FUNCTION_BLOCK EM_Utilities EXTENDS EM_Base IMPLEMENTS I_EM_Utilities
VAR
	//Control modules
	s_diSafetyOk : FB_DigInput;
	s_diPowerOk : FB_DigInput;
	s_diAirPressureOk : FB_DigInput;

	s_doBeaconLedGreen : FB_DigOutput_2;
	s_doBeaconLedYellow : FB_DigOutput_2;
	s_doBeaconLedRed : FB_DigOutput_2;
	
	//States
	s_bStaSafetyOk : BOOL := FALSE;
	s_bStsPowerOk : BOOL := FALSE;
	s_bStaAirPressureOk : BOOL := FALSE;
	
	//s_bStaError
	s_bStaWarning : BOOL;
	
	s_bExtError : BOOL;
	s_bExtWarning : BOOL;
	s_bExtRunning : BOOL;
	
	//Alarms
	s_fbAlarmHandlerSafetyNotOk : FB_AlarmHandler;
	s_fbAlarmHandlerPowerNotOk : FB_AlarmHandler;
	s_fbAlarmHandlerAirPressureNotOk : FB_AlarmHandler;
	
	s_bErrSafetyNotOk : BOOL;
	s_bErrPowerOk : BOOL;
	s_bErrAirPressureNotOk : BOOL;
	
	//Hmi
	s_fbHmiLedSafetyOk : FB_HmiLed;
	s_fbHmiLedPowerOk : FB_HmiLed;
	s_fbHmiLedAirPressureOk : FB_HmiLed;
	s_fbHmiLedBeaconGreen : FB_HmiLed;
	s_fbHmiLedBeaconYellow : FB_HmiLed;
	s_fbHmiLedBeaconRed : FB_HmiLed;
	
	{warning '#TODO' Het zou beter zijn om dit onder te brengen in de onderstaande control modules}
	s_bHmiForceOutputEnabled : BOOL;
END_VAR

VAR_INPUT
	i_eCtrlState		: E_CtrlState;
END_VAR

VAR_OUTPUT
	q_bStaWarning : BOOL;
END_VAR


SUPER^();

METHOD PROTECTED _m_Alarms : BOOL

IF NOT SUPER^._m_Alarms() THEN
	RETURN;
END_IF

//Set error bits
s_bErrSafetyNotOk S= NOT(s_bStaSafetyOk);
s_bErrPowerOk S= NOT(s_bStsPowerOk);
s_bErrAirPressureNotOk S= NOT(s_bStaAirPressureOk);

// Alarm Handlers
s_fbAlarmHandlerSafetyNotOk(
	i_bStaActive := s_bErrSafetyNotOk,
	i_eAlarmLevel := E_AlarmLevel.Alarm, 
	i_sAlarmText := CONCAT(i_sEmName, ' - Safety not OK'));
	
s_fbAlarmHandlerPowerNotOk(
	i_bStaActive := s_bErrPowerOk, 
	i_eAlarmLevel := E_AlarmLevel.Alarm, 
	i_sAlarmText := CONCAT(i_sEmName, ' - Power supply not OK'));
	
s_fbAlarmHandlerAirPressureNotOk(
	i_bStaActive := s_bErrAirPressureNotOk, 
	i_eAlarmLevel := E_AlarmLevel.Alarm, 
	i_sAlarmText := CONCAT(i_sEmName, ' - Air pressure not OK'));
	
// Reset Errors
s_bErrSafetyNotOk R= i_bCmdReset AND s_bStaSafetyOk;
s_bErrPowerOk R= i_bCmdReset AND s_bStsPowerOk;
s_bErrAirPressureNotOk R= i_bCmdReset AND s_bStaAirPressureOk;

s_bStaError := 
	s_fbAlarmHandlerSafetyNotOk.q_bStaActive
	OR s_fbAlarmHandlerPowerNotOk.q_bStaActive
	OR s_fbAlarmHandlerAirPressureNotOk.q_bStaActive;	
	
s_bStaWarning := FALSE;	
	
_m_Alarms := TRUE;
END_METHOD

METHOD PROTECTED _m_Devices : BOOL

IF NOT SUPER^._m_Devices() THEN
	RETURN;
END_IF

//Control module
s_diSafetyOk();
s_diPowerOk();
s_diAirPressureOk();

s_doBeaconLedGreen.i_bStaOutput := s_bExtRunning;
s_doBeaconLedYellow.i_bStaOutput := s_bExtWarning;
s_doBeaconLedRed.i_bStaOutput := s_bExtError;

s_doBeaconLedGreen(i_eCtrlMode := i_eCtrlMode, i_ref_eCtrlState := i_eCtrlState);
s_doBeaconLedYellow(i_eCtrlMode := i_eCtrlMode, i_ref_eCtrlState := i_eCtrlState);
s_doBeaconLedRed(i_eCtrlMode := i_eCtrlMode, i_ref_eCtrlState := i_eCtrlState);
	
_m_Devices := TRUE;
END_METHOD

METHOD PROTECTED _m_Hmi : BOOL

IF NOT SUPER^._m_Hmi() THEN
	RETURN;
END_IF

//Buttons
//..

//Hmi Leds
s_fbHmiLedSafetyOk(i_bStaLed := s_bStaSafetyOk);
s_fbHmiLedPowerOk(i_bStaLed := s_bStsPowerOk);
s_fbHmiLedAirPressureOk(i_bStaLed := s_bStaAirPressureOk);
s_fbHmiLedBeaconGreen(i_bStaLed := s_bExtRunning);
s_fbHmiLedBeaconYellow(i_bStaLed := s_bExtWarning);
s_fbHmiLedBeaconRed(i_bStaLed := s_bExtError);

_m_Hmi := TRUE;
END_METHOD

METHOD PROTECTED _m_Init : BOOL

IF NOT SUPER^._m_Init() THEN
	RETURN;
END_IF

//Control Modules
s_diSafetyOk.i_stSettings.tmInputDelay := T#1S;
s_diPowerOk.i_stSettings.tmInputDelay := T#1S;
s_diAirPressureOk.i_stSettings.tmInputDelay := T#1S;

s_doBeaconLedGreen.i_stSettings.bCfgDelay := FALSE;
s_doBeaconLedGreen.i_stSettings.tmOutputDelay := T#0S;
s_doBeaconLedYellow.i_stSettings.bCfgDelay := FALSE;
s_doBeaconLedYellow.i_stSettings.tmOutputDelay := T#0S;
s_doBeaconLedRed.i_stSettings.bCfgDelay := FALSE;
s_doBeaconLedRed.i_stSettings.tmOutputDelay := T#0S;

//---------------------------------//	
	
//----------------------------------//	
//Hmi 
s_fbHmiLedSafetyOk.p_bStaVisible := FALSE;
s_fbHmiLedSafetyOk.p_sToHmiDescriptionLed := 'Safety Ok';

s_fbHmiLedPowerOk.p_bStaVisible := FALSE;
s_fbHmiLedPowerOk.p_sToHmiDescriptionLed := 'Power Ok';

s_fbHmiLedAirPressureOk.p_bStaVisible := FALSE;
s_fbHmiLedAirPressureOk.p_sToHmiDescriptionLed := 'Air pressure Ok';

s_fbHmiLedBeaconGreen.p_bStaVisible := FALSE;
s_fbHmiLedBeaconGreen.p_sToHmiDescriptionLed := 'Beacon green led';

s_fbHmiLedBeaconYellow.p_bStaVisible := FALSE;
s_fbHmiLedBeaconYellow.p_sToHmiDescriptionLed := 'Beacon yellow led';

s_fbHmiLedBeaconRed.p_bStaVisible := FALSE;
s_fbHmiLedBeaconRed.p_sToHmiDescriptionLed := 'Beacon red led';
	
_m_Init := TRUE;
END_METHOD

METHOD PROTECTED _m_Inputs : BOOL

IF NOT SUPER^._m_Inputs() THEN
	RETURN;
END_IF

s_bStaSafetyOk := s_diSafetyOk.p_bStaInputDelayed AND s_diSafetyOk.p_bStaInput; //on-delay only
s_bStsPowerOk := s_diPowerOk.p_bStaInputDelayed AND s_diPowerOk.p_bStaInput; //on-delay only
s_bStaAirPressureOk := s_diAirPressureOk.p_bStaInputDelayed AND s_diAirPressureOk.p_bStaInput; //on-delay only

_m_Inputs := TRUE;
END_METHOD

METHOD PROTECTED _m_Outputs : BOOL

IF NOT SUPER^._m_Outputs() THEN
	RETURN;
END_IF

s_doBeaconLedGreen.i_bStaOutput := s_bExtRunning;
s_doBeaconLedYellow.i_bStaOutput := s_bExtWarning;
s_doBeaconLedRed.i_bStaOutput := s_bExtError;

q_bStaWarning := s_bStaWarning;

_m_Outputs := TRUE;
END_METHOD

METHOD PUBLIC m_GetGeneralState : BOOL
VAR_INPUT
	i_bError : BOOL;
	i_bWarning : BOOL;
	i_bRunning : BOOL;
END_VAR

s_bExtError := i_bError;
s_bExtWarning := i_bWarning;
s_bExtRunning := i_bRunning;
END_METHOD

METHOD PUBLIC m_Main : BOOL

IF NOT SUPER^.m_Main() THEN
	RETURN;
END_IF

CASE i_eCtrlMode OF
	E_CtrlMode.IDLE:
		;//Nothing
		
	E_CtrlMode.AUTOMATIC:
		//Execute automatic control (based on request from higher-layer unit)
		;//Nothing
		
	E_CtrlMode.MANUAL:
		//Execute manaual control (based on HMI buttons)
		;//Nothing
		
	E_CtrlMode.MAINTENANCE:
		//Execute maintenance control (HMI control module buttons)
		;//Nothing
	
	E_CtrlMode.IO:
		//Execute IO-test control (HMI output force control)
		; 	//IO-Test control is implemented in lower-layer control modules
		
	E_CtrlMode.CLEANING:
		//Execute cleaning control (cleaning  specific functionalities)
		;	//Cleaning control is not implemented, this could be a done in the future if neccesary
END_CASE

//AUTOMATIC-mode //////////////////////////////////////////////////////////////////////////////////
//..

//MANUAL-mode /////////////////////////////////////////////////////////////////////////////////////
//..

//MAINTENANCE-mode ////////////////////////////////////////////////////////////////////////////////
//..

//IO-mode /////////////////////////////////////////////////////////////////////////////////////////
IF (i_eCtrlMode = E_CtrlMode.IO) AND (i_eCtrlState = E_CtrlState.RUNNING) THEN
	s_bHmiForceOutputEnabled := TRUE;
ELSE
	s_bHmiForceOutputEnabled := FALSE;	
END_IF
END_METHOD

PROPERTY PUBLIC p_bStaAirPressureOk : BOOL
GET

p_bStaAirPressureOk := s_bStaAirPressureOk;
END_GET
END_PROPERTY

PROPERTY PUBLIC p_bStaSafetyOk : BOOL
GET

p_bStaSafetyOk := s_bStaSafetyOk;
END_GET
END_PROPERTY

PROPERTY PUBLIC p_bStsPowerOk : BOOL
GET

p_bStsPowerOk := s_bStsPowerOk;
END_GET
END_PROPERTY

END_FUNCTION_BLOCK

(* stored: Version 1.1.0.1, ProductVersion 3.1.4024.12
   POU EM_Utilities: Id {d3bdaf93-23e0-447c-addf-e1fdaa10e5f0}, SpecialFunc None
   Method _m_Alarms: Id {91068a31-fcc6-4281-af61-d7a6e7120f8c}
   Method _m_Devices: Id {97b8a94d-21c8-46ff-ac2c-0f330eabe3be}
   Method _m_Hmi: Id {97417a1d-1af2-4f07-b43b-e4325d410b41}
   Method _m_Init: Id {7f1871a0-83c4-4557-ac15-5a15f84be50f}
   Method _m_Inputs: Id {458358e5-23ba-4231-abac-3325a6a209a2}
   Method _m_Outputs: Id {535a3bcf-7515-4ea2-9150-50d7560b683c}
   Method m_GetGeneralState: Id {c779e9cb-e8a4-4825-ad08-77e95827b039}
   Method m_Main: Id {6ee57644-97c7-4cd8-ab66-2c7443d8efae}
   Property p_bStaAirPressureOk: Id {0af5c43c-8953-4fa1-af7f-5b3f4e44e13a}
   Get Get: Id {4dede668-7bed-49aa-adc6-f4d7ad59be53}
   Property p_bStaSafetyOk: Id {7ea03187-b7ec-46c2-a694-807e2d1d70bb}
   Get Get: Id {7f5e3440-eaae-47cd-8f92-6961cd1007ef}
   Property p_bStsPowerOk: Id {4313e908-4780-46b5-aee4-16ddce14fbff}
   Get Get: Id {b2a078c1-b0bd-4ba8-8232-d29d32a14d28} *)
